(* LS Electric XG5000 project: OUTFULLS *)
(* PLC LSPLC *)

PROGRAM NewProgram (* task: 스캔 프로그램 *)

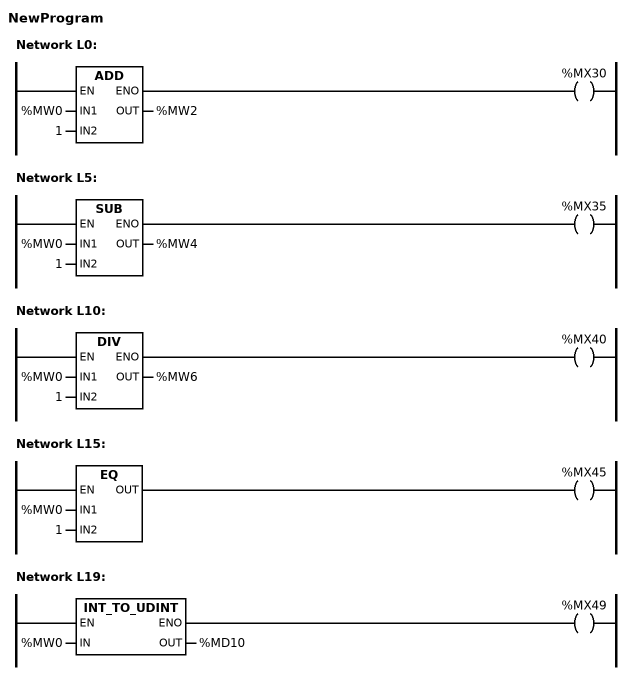
(* Rung L0 *)
%MW2 := %MW0 + 1;
%MX30 := TRUE;
(* Rung L5 *)
%MW4 := %MW0 - 1;
%MX35 := TRUE;
(* Rung L10 *)
%MW6 := %MW0 / 1;
%MX40 := TRUE;
(* Rung L15 *)
%MX45 := %MW0 = 1;
(* Rung L19 *)
%MD10 := INT_TO_UDINT(%MW0);
%MX49 := TRUE;
END_PROGRAM